{attribute 'linkalways'} 
{attribute 'no_explicit_call' := 'This FB is a CLASS and must be accessed using methods or properties'}
{attribute 'enable_dynamic_creation'}
FUNCTION_BLOCK Datatypes IMPLEMENTS I_Datatypes
VAR
	eventEmitter : EventEmitter;
	primitives : Dictionary;
	structures : Dictionary;
	alias : Dictionary;
END_VAR

METHOD PUBLIC Accept
VAR_INPUT
	Visitor : I_DatatypeVisitor;
END_VAR
AcceptPrimative(Visitor);
AcceptStructures(Visitor);
AcceptAlias(Visitor);
END_METHOD

METHOD PRIVATE AcceptAlias
VAR_INPUT
	Visitor : I_DatatypeVisitor;
END_VAR
VAR
	enumerator : I_ForwardEnumerator;
	datatype : I_Datatype;
END_VAR
enumerator := alias.GetEnumerator();

WHILE (enumerator.MoveNext()) DO
	IF enumerator.TryGet(datatype) THEN
		datatype.Accept(Visitor);
	END_IF
END_WHILE

enumerator.Dispose();
END_METHOD

METHOD PRIVATE AcceptPrimative
VAR_INPUT
	Visitor : I_DatatypeVisitor;
END_VAR
VAR
	enumerator : I_ForwardEnumerator;
	datatype : I_Datatype;
END_VAR
enumerator := primitives.GetEnumerator();

WHILE (enumerator.MoveNext()) DO
	IF enumerator.TryGet(datatype) THEN
		datatype.Accept(Visitor);
	END_IF
END_WHILE

enumerator.Dispose();
END_METHOD

METHOD PRIVATE AcceptStructures
VAR_INPUT
	Visitor : I_DatatypeVisitor;
END_VAR
VAR
	enumerator : I_ForwardEnumerator;
	datatype : I_Datatype;
END_VAR
enumerator := structures.GetEnumerator();

WHILE (enumerator.MoveNext()) DO	
	IF enumerator.TryGet(datatype) THEN
		datatype.Accept(Visitor);
	END_IF
END_WHILE

enumerator.Dispose();
END_METHOD

METHOD PROTECTED EmitOnAliasDatatypeAddedEvent
VAR_INPUT
	Datatype : I_AliasDatatype;
END_VAR
VAR
	pAliasDatatypeAddedEvent : POINTER TO AliasDatatypeAddedEvent;
END_VAR
pAliasDatatypeAddedEvent := __NEW(AliasDatatypeAddedEvent(Target := Datatype));
eventEmitter.Emit('OnDatatypeAdded',pAliasDatatypeAddedEvent^);
pAliasDatatypeAddedEvent^.Dispose();
END_METHOD

METHOD PROTECTED EmitOnDatatypeAddedEvent
VAR_INPUT
	Datatype : I_Datatype;
END_VAR
VAR
	pDatatypeAddedEvent : POINTER TO DatatypeAddedEvent;
END_VAR
pDatatypeAddedEvent := __NEW(DatatypeAddedEvent(Target := Datatype));
eventEmitter.Emit('OnDatatypeAdded',pDatatypeAddedEvent^);
pDatatypeAddedEvent^.Dispose();
END_METHOD

METHOD PROTECTED EmitOnStructuredDatatypeAddedEvent
VAR_INPUT
	Datatype : I_StructuredDatatype;
END_VAR
VAR
	pStructuredDatatypeAddedEvent : POINTER TO StructuredDatatypeAddedEvent;
END_VAR
pStructuredDatatypeAddedEvent := __NEW(StructuredDatatypeAddedEvent(Target := Datatype));
eventEmitter.Emit('OnDatatypeAdded',pStructuredDatatypeAddedEvent^);
pStructuredDatatypeAddedEvent^.Dispose();
END_METHOD

METHOD PUBLIC GetAliasByIdentifier : BOOL
VAR_INPUT
	Identifier : T_MAXSTRING;
	Destination : REFERENCE TO I_AliasDatatype;
END_VAR
GetAliasByIdentifier := alias.TryGetValue(Identifier, Destination);
END_METHOD

METHOD PUBLIC GetPrimitiveByIecType : BOOL
VAR_INPUT
	Identifier : T_MAXSTRING;
	Destination : REFERENCE TO I_AliasDatatype;
END_VAR
GetPrimitiveByIecType := primitives.TryGetValue(Identifier, Destination);
END_METHOD

METHOD PUBLIC GetStructureByIdentifier : BOOL
VAR_INPUT
	Identifier : T_MAXSTRING;
	Destination : REFERENCE TO I_StructuredDatatype;
END_VAR
GetStructureByIdentifier := structures.TryGetValue(Identifier, Destination);
END_METHOD

METHOD PUBLIC OffEvent
VAR_INPUT
	EventName : T_MaxString;
	EventHandler : I_EventHandler;
END_VAR
eventEmitter.OffEvent(EventName, EventHandler);
END_METHOD

METHOD PUBLIC OnceEvent
VAR_INPUT
	EventName : T_MaxString;
	EventHandler : I_EventHandler;
END_VAR
eventEmitter.OnceEvent(EventName, EventHandler);
END_METHOD

METHOD PUBLIC OnEvent
VAR_INPUT
	EventName : T_MaxString;
	EventHandler : I_EventHandler;
END_VAR
eventEmitter.OnEvent(EventName, EventHandler);
END_METHOD

METHOD RegisterDatatype
VAR_INPUT
	Datatype : I_Datatype;
END_VAR
VAR
	datatypeAsStructure : I_StructuredDatatype;
	datatypeAsAlias : I_AliasDatatype;
END_VAR
IF Datatype.TryResolveAsStructuredType(datatypeAsStructure) THEN
	structures.AddOrUpdate(datatypeAsStructure.Identifier, datatypeAsStructure);
	emitOnStructuredDatatypeAddedEvent(datatypeAsStructure);
	RETURN;
END_IF

IF Datatype.TryResolveAsAliasType(datatypeAsAlias) THEN
	alias.AddOrUpdate(datatypeAsAlias.Identifier, datatypeAsAlias);
	emitOnAliasDatatypeAddedEvent(datatypeAsAlias);
	RETURN;
END_IF

// add enumeration

// add arrays

primitives.AddOrUpdate(Datatype.IecType, Datatype);
emitOnDatatypeAddedEvent(Datatype);
END_METHOD

METHOD PRIVATE SerializeAliasTypeWith
VAR_INPUT
	Serializer : I_Serializer;
END_VAR
VAR
	enumerator : I_ForwardEnumerator;
	datatype : I_AliasDatatype;
END_VAR
enumerator := alias.GetEnumerator();

WHILE enumerator.MoveNext() DO
	IF enumerator.TryGet(datatype) THEN
		datatype.SerializeTypeWith(Serializer);
	END_IF
END_WHILE

enumerator.Dispose();
END_METHOD

METHOD PRIVATE SerializePrimitiveTypeWith
VAR_INPUT
	Serializer : I_Serializer;
END_VAR
VAR
	enumerator : I_ForwardEnumerator;
	datatype : I_Datatype;
END_VAR
enumerator := primitives.GetEnumerator();

WHILE enumerator.MoveNext() DO
	IF enumerator.TryGet(datatype) THEN
		datatype.SerializeTypeWith(Serializer);
	END_IF
END_WHILE

enumerator.Dispose();
END_METHOD

METHOD PRIVATE SerializeStructuresTypeWith
VAR_INPUT
	Serializer : I_Serializer;
END_VAR
VAR
	enumerator : I_ForwardEnumerator;
	datatype : I_StructuredDatatype;
END_VAR
enumerator := structures.GetEnumerator();

WHILE enumerator.MoveNext() DO
	IF enumerator.TryGet(datatype) THEN
		datatype.SerializeTypeWith(Serializer);
	END_IF
END_WHILE

enumerator.Dispose();
END_METHOD

METHOD PUBLIC SerializeTypeWith
VAR_INPUT
	Serializer : I_Serializer;
END_VAR
Serializer.StartObject();
Serializer.AddKey('datatypes');
Serializer.StartArray();
SerializePrimitiveTypeWith(Serializer);
SerializeStructuresTypeWith(Serializer);
SerializeAliasTypeWith(Serializer);
Serializer.EndArray();
Serializer.EndObject();
END_METHOD

END_FUNCTION_BLOCK

(* stored: Version 1.1.0.1, ProductVersion 3.1.4024.12
   POU Datatypes: Id {6c9601e9-cb69-03bb-11a8-f515550e2ea0}, SpecialFunc None
   Folder Private: Id {78c7fbc9-34a6-07fb-3bc4-4515a5ffd2f8}
   Folder Protected: Id {62284699-e54c-4ace-9c90-cfc00ad6615f}
   Method Accept: Id {fcfbce77-74fe-0e7f-175c-9294ec3c39b4}
   Method AcceptAlias: Id {eebff695-065a-08a1-1e04-8c2f78db7db6}
   Method AcceptPrimative: Id {9bf55bbf-f32f-051d-0f13-603c59d90ff4}
   Method AcceptStructures: Id {0be83cdd-9f3d-006f-168a-32f0dcd2ea1b}
   Method EmitOnAliasDatatypeAddedEvent: Id {48f3f8c0-b856-06c2-1476-2275e86601d0}
   Method EmitOnDatatypeAddedEvent: Id {f5aee9fa-149f-4d4a-941b-789f116d8acd}
   Method EmitOnStructuredDatatypeAddedEvent: Id {a18a95cd-9dcd-064f-2299-b1fff04c15e6}
   Method GetAliasByIdentifier: Id {c51a72ba-8246-0912-0373-b9f426726bf5}
   Method GetPrimitiveByIecType: Id {d7c1dc3c-b86e-070f-1acc-07d73621282f}
   Method GetStructureByIdentifier: Id {44d14eb2-6e6f-0c87-2cf3-368078e88ab2}
   Method OffEvent: Id {be08ab23-08fb-430a-a77c-ca6a54a7087c}
   Method OnceEvent: Id {4426e051-4462-487d-a90d-644adbd72798}
   Method OnEvent: Id {9f41dac2-39fa-4d7e-b411-26a1d65961d8}
   Method RegisterDatatype: Id {8eb94590-4376-0771-0495-507ce775abe7}
   Method SerializeAliasTypeWith: Id {6d9005d4-2c94-0000-344a-c53fded1d5e3}
   Method SerializePrimitiveTypeWith: Id {fe87a4d8-360d-05d5-0318-5f7f98007760}
   Method SerializeStructuresTypeWith: Id {7706e606-9daa-0b93-01d0-f079e5c509d2}
   Method SerializeTypeWith: Id {11dc85a9-60d6-087d-1a5a-82b29db26b01} *)
